// SIMATIC S7-200 project (STEP 7-Micro/WIN), CPU 224 REL 02.01

ORGANIZATION_BLOCK MAIN:OB1
TITLE=程序注释
BEGIN
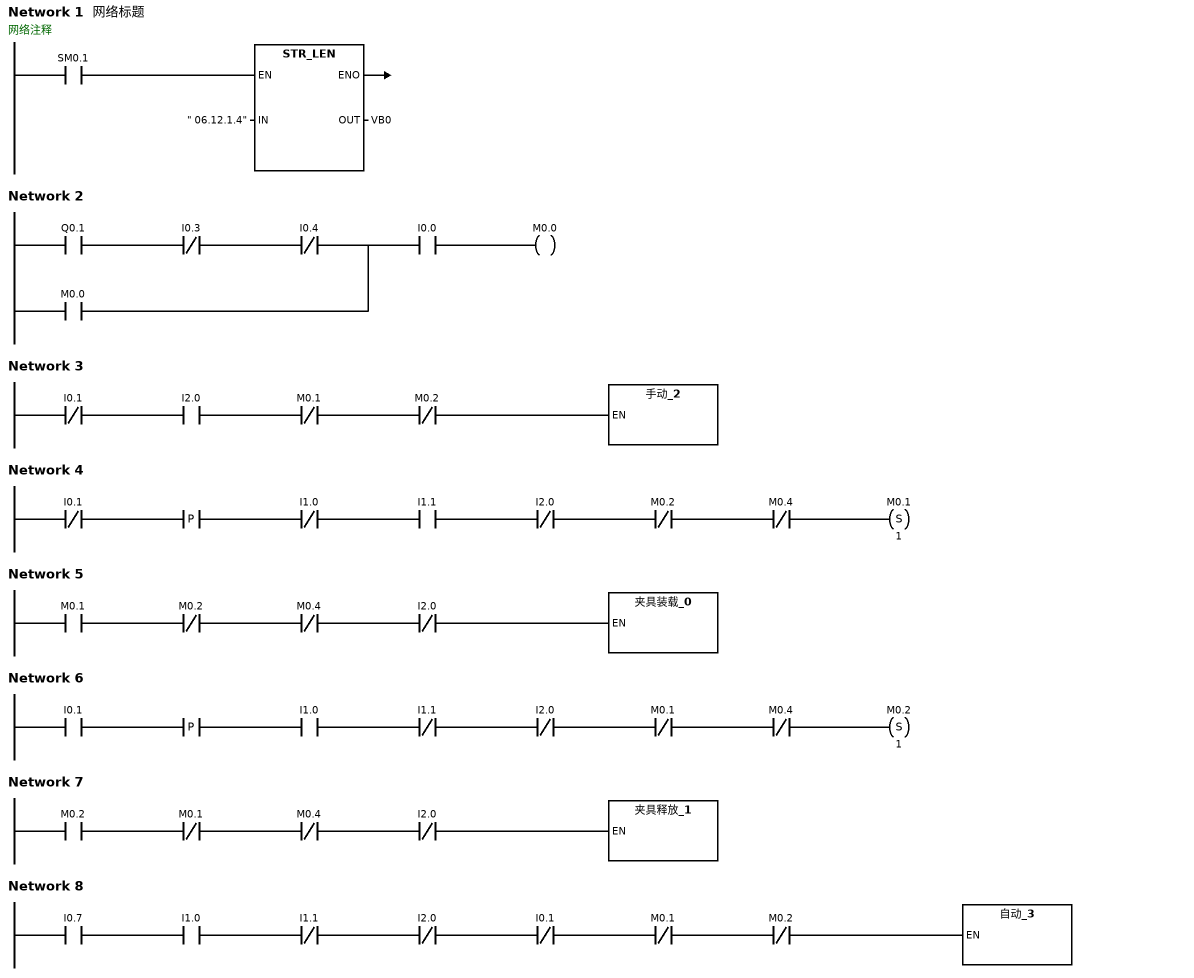
Network 1 // 网络标题
// 网络注释
LD     SM0.1
SLEN   " 06.12.1.4", VB0
Network 2
LD     Q0.1
AN     I0.3
AN     I0.4
O      M0.0
A      I0.0
=      M0.0
Network 3
LDN    I0.1
A      I2.0
AN     M0.1
AN     M0.2
CALL   手动_2:SBR2
Network 4
LDN    I0.1
EU
AN     I1.0
A      I1.1
AN     I2.0
AN     M0.2
AN     M0.4
S      M0.1, 1
Network 5
LD     M0.1
AN     M0.2
AN     M0.4
AN     I2.0
CALL   夹具装载_0:SBR0
Network 6
LD     I0.1
EU
A      I1.0
AN     I1.1
AN     I2.0
AN     M0.1
AN     M0.4
S      M0.2, 1
Network 7
LD     M0.2
AN     M0.1
AN     M0.4
AN     I2.0
CALL   夹具释放_1:SBR1
Network 8
LD     I0.7
A      I1.0
AN     I1.1
AN     I2.0
AN     I0.1
AN     M0.1
AN     M0.2
CALL   自动_3:SBR3
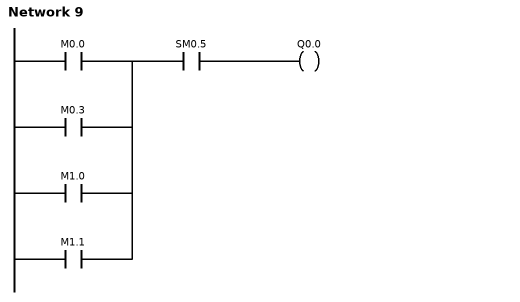
Network 9
LD     M0.0
O      M0.3
O      M1.0
O      M1.1
A      SM0.5
=      Q0.0
END_ORGANIZATION_BLOCK

// SBR0: protected block, not included

// SBR1: protected block, not included

// SBR2: protected block, not included

// SBR3: protected block, not included

// SBR4: protected block, not included

// INT0: protected block, not included
